(*

.. <legal notes>

legal notes
=================
| SPDX-FileCopyrightText: © 2026 Oleksandr Tiutyk <trofimich@gmail.com>
| SPDX-License-Identifier: LGPL-3.0-only
| For details check: LGPL-3.0-only_

.. _LGPL-3.0-only: https://www.gnu.org/licenses/lgpl-3.0.en.html

.. </legal notes>

*)

FUNCTION_BLOCK ABSTRACT AutomationController 
VAR_GENERIC CONSTANT
	{attribute 'hide'} 
    _ChildCount : Core.INT_LENGTH := 0;
END_VAR
EXTENDS AutomationComponent IMPLEMENTS IAutomationController
VAR
	{attribute 'hide'} 
	_Plugins : POINTER TO IAutomationControllerPlugin;
	{attribute 'hide'} 
	_PluginCount : Core.INT_LENGTH;
END_VAR

METHOD PROTECTED FINAL AssingPlugins 
VAR_INPUT
	plugins : ARRAY [*] OF IAutomationControllerPlugin;
END_VAR
_Plugins := plugins;

IF plugins <> 0 THEN
	_PluginCount := TO_INT(1 + UPPER_BOUND(plugins, 1) - LOWER_BOUND(plugins, 1));
ELSE
	_PluginCount := 0;
END_IF
END_METHOD

{attribute 'monitoring' := 'call'}
PROPERTY FINAL ChildCount : Core.INT_LENGTH
GET
ChildCount := _ChildCount;
END_GET
END_PROPERTY

{attribute 'monitoring' := 'call'}
PROPERTY ABSTRACT Children : REFERENCE TO ARRAY [0.._ChildCount - 1] OF IChildAutomationComponent
GET
END_GET
END_PROPERTY

PROPERTY PROTECTED FINAL InternalChildCount : Core.INT_INDEX
GET
InternalChildCount := _ChildCount;
END_GET
END_PROPERTY

METHOD PROTECTED FINAL InternalTryGetChildByIndex : IChildAutomationComponent
VAR_INPUT
	index : Core.INT_INDEX;
END_VAR
IF __ISVALIDREF(Children) AND_THEN index >= 0 AND_THEN index <= _ChildCount THEN
	InternalTryGetChildByIndex := Children[index];
END_IF
END_METHOD

METHOD PROTECTED OnAfterDevicesProcessInput
END_METHOD

METHOD PROTECTED OnAfterDevicesProcessOutput
END_METHOD

METHOD PROTECTED FINAL OnAfterExecute
VAR
	exceptionCode : __SYSTEM.ExceptionCode;
	exception : Core.IException;	
	exceptionHandlingResult : PROBLEM_HANDLING_RESULT;

	i : Core.INT_INDEX;
	
	child : IChildAutomationComponent;
	
	plugin : IAutomationControllerPlugin;
	
	outputDevice : IOutputDevice;	
END_VAR
__TRY
	OnBeforeDevicesProcessOutput();
__CATCH(exceptionCode)		
	exception := Core.ExceptionManager.GetLastException(exceptionCode);
					
	exceptionHandlingResult := OnHandleException(exception, EXCEPTION_CATCH_POINT.ON_BEFORE_CHILDREN_PROCESS_OUTPUT);

	ProcessException(exception, exceptionHandlingResult, "OnBeforeDevicesProcessOutput error");
__ENDTRY

FOR i := 0 TO ChildCount - 1 DO
	child := InternalTryGetChildByIndex(i);
	
	IF NOT child.Enabled OR_ELSE NOT __QUERYINTERFACE(child, outputDevice) THEN
		CONTINUE;
	END_IF

	outputDevice.ProcessOutput(); 
	
	IF outputDevice.HasError AND_THEN outputDevice.Error.Severity = Core.ERROR_SEVERITY.CRITICAL THEN
		exceptionHandlingResult := OnHandleChildCriticalError(outputDevice);
		
		ProcessChildError(outputDevice.Error, exceptionHandlingResult, Core.WideStrings.Concat255("Child[", TO_WSTRING(i), "(", outputDevice.Name, ")].ProcessOutput error"));
	END_IF
END_FOR

__TRY
	OnAfterDevicesProcessOutput();
__CATCH(exceptionCode)		
	exception := Core.ExceptionManager.GetLastException(exceptionCode);
					
	exceptionHandlingResult := OnHandleException(exception, EXCEPTION_CATCH_POINT.ON_AFTER_CHILDREN_PROCESS_OUTPUT);

	ProcessException(exception, exceptionHandlingResult, "OnAfterDevicesProcessOutput error");
__ENDTRY

FOR i := 0 TO PluginCount - 1 DO
	plugin := TryGetPluginByIndex(i);
	
	IF plugin <> 0 THEN
		__TRY
			plugin.OnAfterControllerExecute(THIS^);
		__CATCH(exceptionCode)		
			exception := Core.ExceptionManager.GetLastException(exceptionCode);
							
			exceptionHandlingResult := OnHandleException(exception, EXCEPTION_CATCH_POINT.ON_AFTER_EXECUTE_PLUGINS);
		
			ProcessException(exception, exceptionHandlingResult, Core.WideStrings.Concat255("plugin[", TO_WSTRING(i), "].OnAfterControllerExecute error"));
		__ENDTRY		
	END_IF
END_FOR
END_METHOD

METHOD PROTECTED OnBeforeChildrenInitializing
VAR
	devicesNotSpecifiedException : Core.DataMemberNotSpecifiedException;
END_VAR
IF _ChildCount > 0 AND_THEN NOT __ISVALIDREF(Children) THEN
	devicesNotSpecifiedException.ThrowByObject(THIS^, __POUNAME(), __POSITION(), 'Children');
END_IF
END_METHOD

METHOD PROTECTED OnBeforeDevicesProcessInput
END_METHOD

METHOD PROTECTED OnBeforeDevicesProcessOutput
END_METHOD

METHOD PROTECTED FINAL OnBeforeExecute
VAR
	exceptionCode : __SYSTEM.ExceptionCode;
	exception : Core.IException;	
	exceptionHandlingResult : PROBLEM_HANDLING_RESULT;

	i : Core.INT_INDEX;

	child : IChildAutomationComponent;
	
	plugin : IAutomationControllerPlugin;
	
	inputDevice : IInputDevice;
END_VAR
FOR i := 0 TO PluginCount - 1 DO
	plugin := TryGetPluginByIndex(i);
	
	IF plugin <> 0 THEN
		__TRY
			plugin.OnBeforeControllerExecute(THIS^);
		__CATCH(exceptionCode)		
			exception := Core.ExceptionManager.GetLastException(exceptionCode);
							
			exceptionHandlingResult := OnHandleException(exception, EXCEPTION_CATCH_POINT.ON_BEFORE_EXECUTE_PLUGINS);
		
			ProcessException(exception, exceptionHandlingResult, Core.WideStrings.Concat255("plugin[", TO_WSTRING(i), "].OnBeforeControllerExecute error"));
		__ENDTRY		
	END_IF
END_FOR

__TRY
	OnBeforeDevicesProcessInput();
__CATCH(exceptionCode)		
	exception := Core.ExceptionManager.GetLastException(exceptionCode);
					
	exceptionHandlingResult := OnHandleException(exception, EXCEPTION_CATCH_POINT.ON_BEFORE_CHILDREN_PROCESS_INPUT);

	ProcessException(exception, exceptionHandlingResult, "OnBeforeDevicesProcessInput error");
__ENDTRY

FOR i := 0 TO ChildCount - 1 DO
	child := InternalTryGetChildByIndex(i);

	IF NOT child.Enabled OR_ELSE NOT __QUERYINTERFACE(child, inputDevice) THEN
		CONTINUE;
	END_IF

	inputDevice.ProcessInput(); 

	IF inputDevice.HasError AND_THEN inputDevice.Error.Severity = Core.ERROR_SEVERITY.CRITICAL THEN
		exceptionHandlingResult := OnHandleChildCriticalError(inputDevice);
		
		ProcessChildError(inputDevice.Error, exceptionHandlingResult, Core.WideStrings.Concat255("Child[", TO_WSTRING(i), "(", inputDevice.Name, ")].ProcessInput error"));
	END_IF	
END_FOR

__TRY
	OnAfterDevicesProcessInput();
__CATCH(exceptionCode)		
	exception := Core.ExceptionManager.GetLastException(exceptionCode);
					
	exceptionHandlingResult := OnHandleException(exception, EXCEPTION_CATCH_POINT.ON_AFTER_CHILDREN_PROCESS_INPUT);

	ProcessException(exception, exceptionHandlingResult, "OnAfterDevicesProcessInput error");
__ENDTRY
END_METHOD

{attribute 'monitoring' := 'call'}
PROPERTY FINAL PluginCount : Core.INT_LENGTH
GET
PluginCount := _PluginCount;
END_GET
END_PROPERTY

METHOD FINAL TryGetChildByIndex : IChildAutomationComponent
VAR_INPUT
	index : Core.INT_INDEX;
END_VAR
TryGetChildByIndex := InternalTryGetChildByIndex(index);
END_METHOD

METHOD TryGetPluginByIndex : IAutomationControllerPlugin
VAR_INPUT
	index : Core.INT_INDEX;
END_VAR
IF _PluginCount > index THEN
	TryGetPluginByIndex := _Plugins[index];
END_IF
END_METHOD

END_FUNCTION_BLOCK

(* stored: Version 1.1.0.1
   POU AutomationController: Id {6b707d9d-36a1-4196-b85e-da052ddd92c8}, SpecialFunc None
   Folder Methods to override: Id {6ec9b840-4a77-44e7-8c31-53666e455ae9}
   Folder ProcessInput: Id {f88db65f-7256-4f0b-903f-ce2776a2a205}
   Folder ProcessOutput: Id {5f362344-8bb9-467e-b80b-e33887713368}
   Folder Overriden members: Id {c5ec7856-9826-474b-a801-c545bcc0d575}
   Method AssingPlugins: Id {898fe1ab-4afc-4d2c-b446-7bee770fabf4}
   Property ChildCount: Id {9220f711-cd6b-4535-afb7-2d29bd70dbf0}
   Get Get: Id {7ecd62bb-cc61-4886-a3b7-812711794d0b}
   Property Children: Id {b6d998b9-573d-4770-83de-0928458fcc43}
   Get Get: Id {b6ba42f9-ee1b-4d18-84e7-5d5ae248c53f}
   Property InternalChildCount: Id {bd3bcc14-1030-4962-be44-0b94cffa3f06}
   Get Get: Id {30029f6a-e588-4d91-93d3-d543769e010b}
   Method InternalTryGetChildByIndex: Id {9ada9ba3-31c5-480e-8ac0-dd147a83c6f4}
   Method OnAfterDevicesProcessInput: Id {ead89ebd-a27d-432f-966e-e687aaaba46d}
   Method OnAfterDevicesProcessOutput: Id {6bf5950d-bcab-4e58-9158-847d05b05354}
   Method OnAfterExecute: Id {c5f93a76-dee4-4362-8224-f58ff2acf349}
   Method OnBeforeChildrenInitializing: Id {96a6f588-939f-4fde-a4b8-d8f2002a7ef4}
   Method OnBeforeDevicesProcessInput: Id {b8dd0ed9-825b-4f71-845c-b8b9e8809df1}
   Method OnBeforeDevicesProcessOutput: Id {4c45b535-4195-4589-898d-c477e10dcef0}
   Method OnBeforeExecute: Id {ce282655-acf4-4ac1-8632-e5d04ecfe5cd}
   Property PluginCount: Id {c48dfd84-c0df-4e03-b68e-6081a02a9f8d}
   Get Get: Id {5dc2143c-2fd9-40fa-82bb-d9ba834aa42a}
   Method TryGetChildByIndex: Id {41e536e8-bb48-46c8-b4d8-f8835e391a1a}
   Method TryGetPluginByIndex: Id {b96b6560-7aba-4b72-8158-2ea48dd1ce51} *)
